(* PLC project SafeLOGIC-1, BrAutomation SafeDESIGNER  5.15.0.0 *)
(* stored: companyURL http://www.br-automation.com, creationDateTime Sat Sep 17 18:19:39 2022 *)

PROGRAM Output_Card

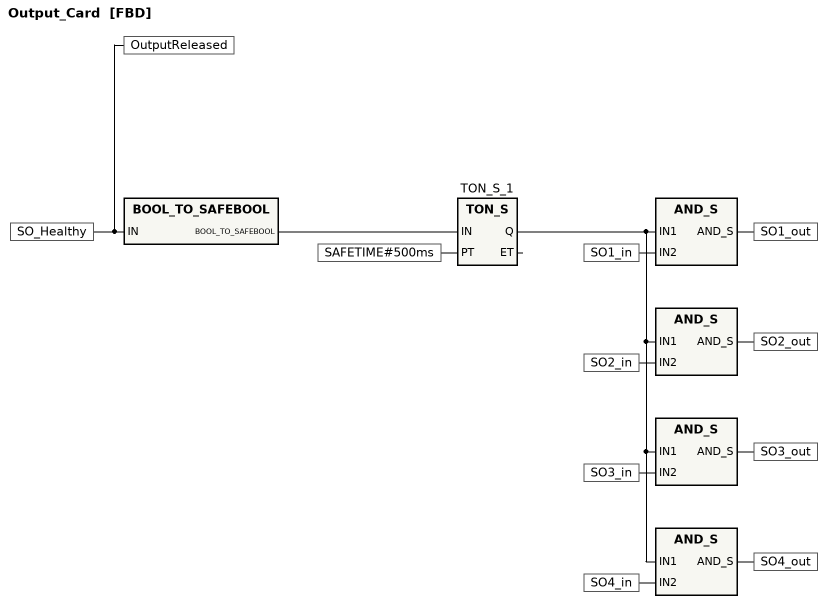
(* FBD diagram, written out as Structured Text *)
OutputReleased := SO_Healthy;
TON_S_1(IN := BOOL_TO_SAFEBOOL(SO_Healthy), PT := SAFETIME#500ms);
SO1_out := AND_S(TON_S_1.Q, SO1_in);
SO2_out := AND_S(TON_S_1.Q, SO2_in);
SO3_out := AND_S(TON_S_1.Q, SO3_in);
SO4_out := AND_S(TON_S_1.Q, SO4_in);
END_PROGRAM
